// TIA Portal project "PPA-Projekt" (V17)
// Projekt do předmětu PPA

(* hardware
DEVICE "S7-1500/ET200MP station_1"  S7-1500 station
   slot 0: "Rail_0"  Rack  6ES7 590-1***0-0AA0
   slot 1: "PLC_1"  CPU 1516-3 PN/DP  6ES7 516-3AN00-0AB0  V1.8
      slot 3: "CPU display_1"  6ES7591-1BA00-0AA0
      slot 32768: "PROFINET interface_1"  X1
         slot 32769: "Port_1"  X1 P1
         slot 32770: "Port_2"  X1 P2
      slot 33024: "PROFINET interface_2"  X2
         slot 33025: "Port_1"  X2 P1
      slot 33280: "DP interface_1"  X3
DEVICE "HMI_1"  KTP700 Basic PN
   slot 0: "HMI_1"  KTP700 Basic PN  6AV2 123-2GB03-0AX0  17.0.0.0
   slot 1: "HMI_RT_1"  KTP700 Basic PN  6AV2 123-2GB03-0AX0  17.0.0.0
   slot 5: "HMI_1.IE_CP_1"  PROFINET Interface  17.0.0.0
      slot 1: "PROFINET Interface_1"  PROFINET Interface
         slot 1: "Port_1"  Port
*)

// ===== PLC "PLC_1"  CPU 1516-3 PN/DP =====

VAR_GLOBAL   // PLC tag table "Default tag table"
   "SystemInput" AT %MW5 : Int;   // Passed value to PID Setpoints
   "Clock_Byte" AT %MB0 : Byte;
   "Clock_10Hz" AT %M0.0 : Bool;
   "Clock_5Hz" AT %M0.1 : Bool;
   "Clock_2.5Hz" AT %M0.2 : Bool;
   "Clock_2Hz" AT %M0.3 : Bool;
   "Clock_1.25Hz" AT %M0.4 : Bool;
   "Clock_1Hz" AT %M0.5 : Bool;
   "Clock_0.625Hz" AT %M0.6 : Bool;
   "Clock_0.5Hz" AT %M0.7 : Bool;
   "System_Byte" AT %MB1 : Byte;
   "FirstScan" AT %M1.0 : Bool;
   "DiagStatusUpdate" AT %M1.1 : Bool;
   "AlwaysTRUE" AT %M1.2 : Bool;
   "AlwaysFALSE" AT %M1.3 : Bool;
   "SwitchInput" AT %M2.0 : Bool;   // Change SetValue at PID inputs
   "SetValue" AT %MW3 : Int;   // SetValue variable
   "Enable_SystemMatlab" AT %M9.0 : Bool;
   "Enable_SystemTia" AT %M9.1 : Bool;
END_VAR

DATA_BLOCK "LSIM_Matlab"   // DB1
{ S7_Optimized_Access := 'TRUE' }
VERSION : 2.01
// stored: InstanceOfName LSim_PT2aper
"LSim_PT2aper"
BEGIN
END_DATA_BLOCK

DATA_BLOCK "LSIM_TIA"   // DB6
{ S7_Optimized_Access := 'TRUE' }
VERSION : 2.01
// stored: InstanceOfName LSim_PT2aper_1
"LSim_PT2aper_1"
BEGIN
END_DATA_BLOCK

FUNCTION_BLOCK "LSim_PT2aper"   // FB53, SCL
{ S7_Optimized_Access := 'TRUE' }
VERSION : 2.01
   VAR_INPUT
      calcParam : Bool;   // recalculate with new parameters
      input : Real;   // input signal
      tmLag1 : Real := 2.0;   // time constant T1 [sec]
      tmLag2 : Real := 0.2;   // time constant T2 [sec]
      gain : Real := 1.0;   // gain factor
      cycle : Real := 0.1;   // cyclic time [sec]
      maxOut : Real := 100.0;   // max. output limit
      minOut : Real;   // min. output limit
      reset : Bool;   // resets all relevant parameters to ‘0’ including the output
   END_VAR
   VAR_OUTPUT
      error : Bool;   // error (#tmLag1 <= 0 or #tmLag2 <= 0 or #tmLag1 = #tmLag2)
      status : Word;   // status (if #error = TRUE then status = 16#8001)
      maxReached : Bool;   // output has reached max. limit
      minReached : Bool;   // output has reached min. limit
      output : Real;   // output signal (if #error = FALSE)
   END_VAR
   VAR
      statRxn2 : Real;   // delayed input signal (n-2)
      statRxn1 : Real;   // delayed input signal (n-1)
      statRyn2 : Real;   // delayed output signal (n-2)
      statRyn1 : Real;   // delayed output signal (n-1)
      statRf1 : Real;
      statRf2 : Real;
      statRe1 : Real;
      statRe2 : Real;
      statAlpha : Real;
      statBeta : Real;
      statGamma : Real;
      statDelta : Real;
      statOverfirst : Bool;
      statOutput : Real;   // Output signal
   END_VAR
BEGIN
   //=============================================================================
   //SIEMENS AG
   //(c)Copyright 2017 All Rights Reserved
   //-----------------------------------------------------------------------------
   //Library:       Library for Controlled System Simulation
   //Tested with:   S7-1500 FW V2.0 / S7-1200 FW V4.2
   //Engineering:   STEP 7 V14 Upd2 (TIA Portal)
   //Restrictions:  Cyclic interrupt
   //Requirements:  memory card needed for S7-1500
   //Functionality: Simulation of a aperiodic PT2-System
   //  
   //                    gain
   //  F(p) = -----------------------------
   //         (tmLag1*p + 1)*(tmLag2*p + 1)
   //         
   //  Call the simulation in a cyclic interrupt with
   //  cyclic interrupt time at least = tmLag1/10!
   //-----------------------------------------------------------------------------
   //Change log table:
   //Version  Date       Expert in charge                Changes applied
   //02.00.00 03.02.2016 Siemens Industry Online Support Release (STEP 7 V13 SP1)
   //02.00.01 02.03.2017 Siemens Industry Online Support Release (STEP 7 V14)
   //=============================================================================

   // check parameter
   IF #tmLag1 <= 0 OR #tmLag2 <= 0 OR #tmLag1 = #tmLag2 THEN
     #error := TRUE;
     #status := W#16#8001;     // Parameter Error
     #statRxn1 := 0.0;
     #statRyn1 := 0.0;
     #statRxn2 := 0.0;
     #statRyn2 := 0.0;
     #statOutput := 0;
     #output := 0;
     RETURN;
   ELSE
     #error := FALSE;
     #status := W#16#0000;     // no error
   END_IF;

   // calculates the z-parameter for the difference equatation
   IF #calcParam = True OR NOT #statOverfirst THEN
     #statOverfirst := 1;
     // Calculate z-parameters for IT1-System
     #statAlpha := EXP(- #cycle / #tmLag1);
     #statBeta := EXP(- #cycle / #tmLag2);
     #statGamma := #tmLag1 / (#tmLag1 - #tmLag2);
     #statDelta := #tmLag2 / (#tmLag1 - #tmLag2);
     #statRe1 := - #statAlpha - #statBeta;
     #statRe2 := #statAlpha * #statBeta;
     #statRf1 := #gain * (1 - #statGamma * #statAlpha + #statDelta * #statBeta);
     #statRf2 := #gain * (#statAlpha * #statBeta - #statGamma * #statBeta + #statAlpha * #statDelta);
   END_IF;

   // reset Memory
   IF #reset = True THEN
     #statRxn1 := 0.0;
     #statRyn1 := 0.0;
     #statRxn2 := 0.0;
     #statRyn2 := 0.0;
     #statOutput := 0;
   END_IF;
   //save delayed input signals
   #statRxn2 := #statRxn1;
   #statRxn1 := #input;

   //save delayed output signals
   #statRyn2:=#statRyn1;
   #statRyn1:= #statOutput;

   // difference equatation of the PT2-System
   #statOutput := #statRxn1* #statRf1 + #statRxn2*#statRf2 - #statRyn1*#statRe1 - #statRyn2*#statRe2;

   // max limit of acutating variable
   IF #statOutput > #maxOut THEN
     #statOutput := #maxOut;
     #maxReached:= True;
   ELSE
     #maxReached := False;
   END_IF;

   // min limit of acutating variable
   IF #statOutput < #minOut THEN
     #statOutput := #minOut;
     #minReached := True;
   ELSE
     #minReached := False;
   END_IF;

   #output := #statOutput;
END_FUNCTION_BLOCK

FUNCTION_BLOCK "LSim_PT2aper_1"   // FB54, SCL
{ S7_Optimized_Access := 'TRUE' }
VERSION : 2.01
   VAR_INPUT
      calcParam : Bool;   // recalculate with new parameters
      input : Real;   // input signal
      tmLag1 : Real := 2.0;   // time constant T1 [sec]
      tmLag2 : Real := 0.2;   // time constant T2 [sec]
      gain : Real := 1.0;   // gain factor
      cycle : Real := 0.1;   // cyclic time [sec]
      maxOut : Real := 100.0;   // max. output limit
      minOut : Real;   // min. output limit
      reset : Bool;   // resets all relevant parameters to ‘0’ including the output
   END_VAR
   VAR_OUTPUT
      error : Bool;   // error (#tmLag1 <= 0 or #tmLag2 <= 0 or #tmLag1 = #tmLag2)
      status : Word;   // status (if #error = TRUE then status = 16#8001)
      maxReached : Bool;   // output has reached max. limit
      minReached : Bool;   // output has reached min. limit
      output : Real;   // output signal (if #error = FALSE)
   END_VAR
   VAR
      statRxn2 : Real;   // delayed input signal (n-2)
      statRxn1 : Real;   // delayed input signal (n-1)
      statRyn2 : Real;   // delayed output signal (n-2)
      statRyn1 : Real;   // delayed output signal (n-1)
      statRf1 : Real;
      statRf2 : Real;
      statRe1 : Real;
      statRe2 : Real;
      statAlpha : Real;
      statBeta : Real;
      statGamma : Real;
      statDelta : Real;
      statOverfirst : Bool;
      statOutput : Real;   // Output signal
   END_VAR
BEGIN
   //=============================================================================
   //SIEMENS AG
   //(c)Copyright 2017 All Rights Reserved
   //-----------------------------------------------------------------------------
   //Library:       Library for Controlled System Simulation
   //Tested with:   S7-1500 FW V2.0 / S7-1200 FW V4.2
   //Engineering:   STEP 7 V14 Upd2 (TIA Portal)
   //Restrictions:  Cyclic interrupt
   //Requirements:  memory card needed for S7-1500
   //Functionality: Simulation of a aperiodic PT2-System
   //  
   //                    gain
   //  F(p) = -----------------------------
   //         (tmLag1*p + 1)*(tmLag2*p + 1)
   //         
   //  Call the simulation in a cyclic interrupt with
   //  cyclic interrupt time at least = tmLag1/10!
   //-----------------------------------------------------------------------------
   //Change log table:
   //Version  Date       Expert in charge                Changes applied
   //02.00.00 03.02.2016 Siemens Industry Online Support Release (STEP 7 V13 SP1)
   //02.00.01 02.03.2017 Siemens Industry Online Support Release (STEP 7 V14)
   //=============================================================================

   // check parameter
   IF #tmLag1 <= 0 OR #tmLag2 <= 0 OR #tmLag1 = #tmLag2 THEN
     #error := TRUE;
     #status := W#16#8001;     // Parameter Error
     #statRxn1 := 0.0;
     #statRyn1 := 0.0;
     #statRxn2 := 0.0;
     #statRyn2 := 0.0;
     #statOutput := 0;
     #output := 0;
     RETURN;
   ELSE
     #error := FALSE;
     #status := W#16#0000;     // no error
   END_IF;

   // calculates the z-parameter for the difference equatation
   IF #calcParam = True OR NOT #statOverfirst THEN
     #statOverfirst := 1;
     // Calculate z-parameters for IT1-System
     #statAlpha := EXP(- #cycle / #tmLag1);
     #statBeta := EXP(- #cycle / #tmLag2);
     #statGamma := #tmLag1 / (#tmLag1 - #tmLag2);
     #statDelta := #tmLag2 / (#tmLag1 - #tmLag2);
     #statRe1 := - #statAlpha - #statBeta;
     #statRe2 := #statAlpha * #statBeta;
     #statRf1 := #gain * (1 - #statGamma * #statAlpha + #statDelta * #statBeta);
     #statRf2 := #gain * (#statAlpha * #statBeta - #statGamma * #statBeta + #statAlpha * #statDelta);
   END_IF;

   // reset Memory
   IF #reset = True THEN
     #statRxn1 := 0.0;
     #statRyn1 := 0.0;
     #statRxn2 := 0.0;
     #statRyn2 := 0.0;
     #statOutput := 0;
   END_IF;
   //save delayed input signals
   #statRxn2 := #statRxn1;
   #statRxn1 := #input;

   //save delayed output signals
   #statRyn2:=#statRyn1;
   #statRyn1:= #statOutput;

   // difference equatation of the PT2-System
   #statOutput := #statRxn1* #statRf1 + #statRxn2*#statRf2 - #statRyn1*#statRe1 - #statRyn2*#statRe2;

   // max limit of acutating variable
   IF #statOutput > #maxOut THEN
     #statOutput := #maxOut;
     #maxReached:= True;
   ELSE
     #maxReached := False;
   END_IF;

   // min limit of acutating variable
   IF #statOutput < #minOut THEN
     #statOutput := #minOut;
     #minReached := True;
   ELSE
     #minReached := False;
   END_IF;

   #output := #statOutput;
END_FUNCTION_BLOCK

ORGANIZATION_BLOCK "Main"   // OB1, LAD, ProgramCycle
TITLE = "Main Program Sweep (Cycle)"
{ S7_Optimized_Access := 'TRUE' }
VERSION : 0.1
   VAR_INPUT
      Initial_Call : Bool;   // Initial call of this OB
      Remanence : Bool;   // =True, if remanent data are available
   END_VAR
BEGIN
END_ORGANIZATION_BLOCK

ORGANIZATION_BLOCK "Interupt - PID"   // OB30, LAD, CyclicInterrupt
{ S7_Optimized_Access := 'TRUE' }
VERSION : 0.1
   VAR_INPUT
      Initial_Call : Bool;   // Initial call of this OB
      Event_Count : Int;   // Events discarded
   END_VAR
BEGIN

REGION Network 1
   // PID controller - Matlab
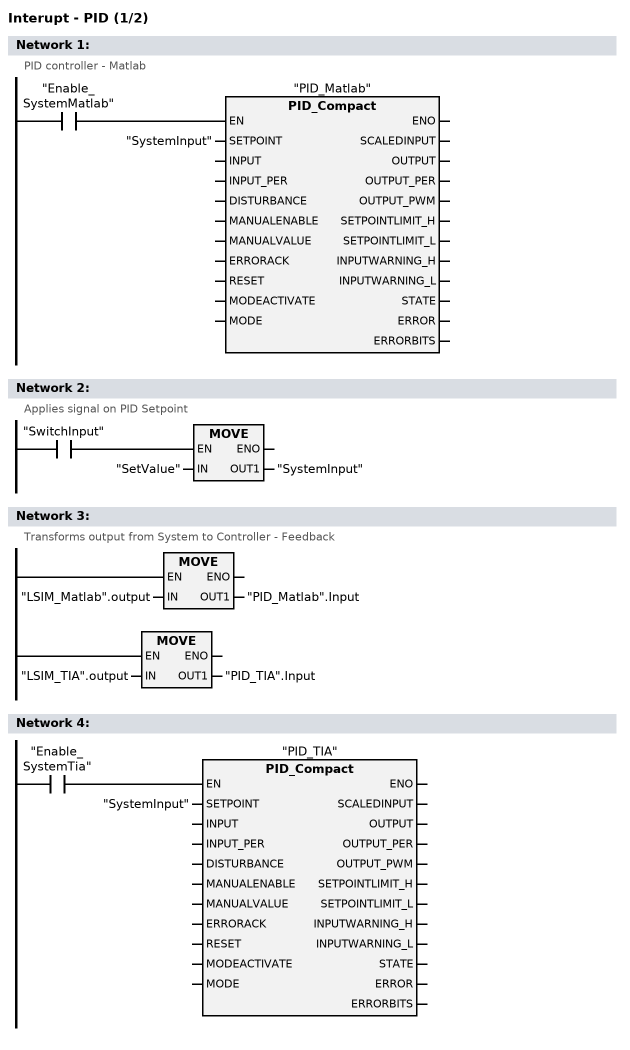
   IF "Enable_SystemMatlab" THEN
       "PID_Matlab"(Setpoint := "SystemInput");   // PID_Compact
   END_IF;
END_REGION

REGION Network 2
   // Applies signal on PID Setpoint
   RUNG wire#powerrail
      Contact( "SwitchInput" )
      Move(in := "SetValue", out1 => "SystemInput")
   END_RUNG
   // the same network as SCL:
   IF "SwitchInput" THEN "SystemInput" := "SetValue"; END_IF;
END_REGION

REGION Network 3
   // Transforms output from System to Controller - Feedback
   RUNG wire#powerrail
      Move(in := "LSIM_Matlab".output, out1 => "PID_Matlab".Input)
   END_RUNG
   RUNG wire#powerrail
      Move(in := "LSIM_TIA".output, out1 => "PID_TIA".Input)
   END_RUNG
   // the same network as SCL:
   "PID_Matlab".Input := "LSIM_Matlab".output;
   "PID_TIA".Input := "LSIM_TIA".output;
END_REGION

REGION Network 4
   IF "Enable_SystemTia" THEN
       "PID_TIA"(Setpoint := "SystemInput");   // PID_Compact
   END_IF;
END_REGION

REGION Network 5
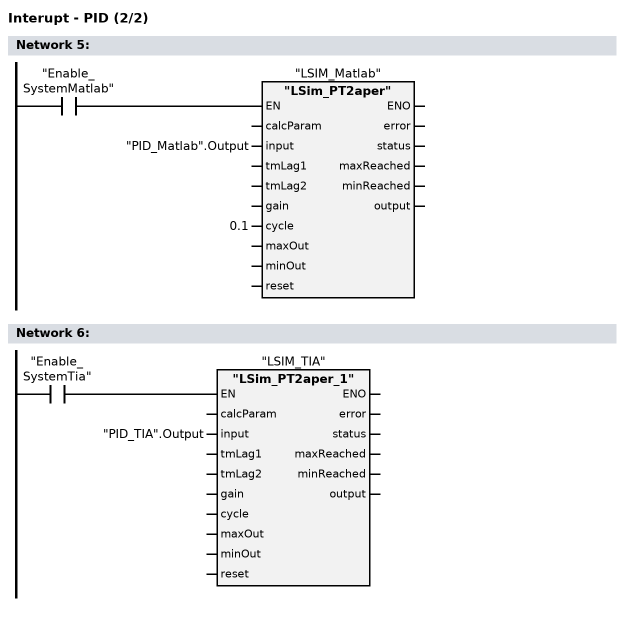
   RUNG wire#powerrail
      Contact( "Enable_SystemMatlab" )
      "LSIM_Matlab"(calcParam :=, input := "PID_Matlab".Output, tmLag1 :=, tmLag2 :=, gain :=, cycle := 0.1, maxOut :=, minOut :=, reset :=, error =>, status =>, maxReached =>, minReached =>, output =>)
   END_RUNG
   // the same network as SCL:
   IF "Enable_SystemMatlab" THEN
       "LSIM_Matlab"(input := "PID_Matlab".Output, cycle := 0.1);   // "LSim_PT2aper"
   END_IF;
END_REGION

REGION Network 6
   RUNG wire#powerrail
      Contact( "Enable_SystemTia" )
      "LSIM_TIA"(calcParam :=, input := "PID_TIA".Output, tmLag1 :=, tmLag2 :=, gain :=, cycle :=, maxOut :=, minOut :=, reset :=, error =>, status =>, maxReached =>, minReached =>, output =>)
   END_RUNG
   // the same network as SCL:
   IF "Enable_SystemTia" THEN
       "LSIM_TIA"(input := "PID_TIA".Output);   // "LSim_PT2aper_1"
   END_IF;
END_REGION
END_ORGANIZATION_BLOCK

ORGANIZATION_BLOCK "Startup"   // OB100, LAD, Startup
TITLE = "Complete Restart"
{ S7_Optimized_Access := 'TRUE' }
VERSION : 0.1
// Intial setup
   VAR_INPUT
      LostRetentive : Bool;   // True if retentive data are lost
      LostRTC : Bool;   // True if date and time are lost
   END_VAR
BEGIN

REGION Network 1
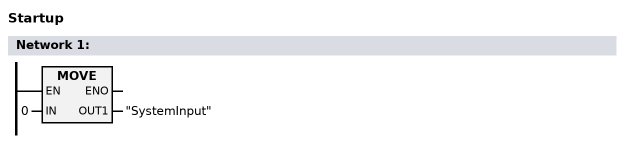
   RUNG wire#powerrail
      Move(in := 0, out1 => "SystemInput")
   END_RUNG
   // the same network as SCL:
   "SystemInput" := 0;
END_REGION
END_ORGANIZATION_BLOCK

(* ===== HMI "HMI_RT_1" =====
system functions are stored by id; their names below are inferred from use
connection "HMI_Connection_1": ETHERNET, SMART_S7_1500_OMS

HMI tags "Default tag table"
   "Tag_ScreenNumber" : UInt, internal
   "LSIM_Matlab_Output" : Real = PLC LSIM_Matlab.output, 100 ms
   "SetValue_Switch" : Bool = PLC SwitchInput AT %M2.0, 100 ms
   "Change_SetValue" : Int = PLC SetValue AT %MW3, 100 ms
   "LSIM_TIA_Output" : Real = PLC LSIM_TIA.output AT %DB1.DBW0, 100 ms
   "System_SetValue" : Int = PLC SystemInput AT %MW5, 100 ms
   "PID_TIA_Output" : Real = PLC PID_TIA.Output, 100 ms
   "PID_Matlab_Output" : Real = PLC PID_Matlab.Output AT %DB1.DBD0, 100 ms
   "Enable_MatlabSystem" : Bool = PLC Enable_SystemMatlab AT %M9.0, 100 ms
   "Enable_TiaSystem" : Bool = PLC Enable_SystemTia AT %M9.1, 100 ms

Template "Template_1" 800x480
   Button "Exit" at 714,429 size 71x50; TextOff 'Exit'; PictureOff "ExitRuntime_KTP700_Basic_PN_TR"; PictureOn "ExitRuntime_KTP700_Basic_PN_TR"
      on Release: StopRuntime(0)
   Button "Template_Button" at 614,429 size 71x50; TextOff 'Text'
   Button "Template_Button_1" at 514,429 size 71x50; TextOff 'Text'
   Button "Template_Button_2" at 414,429 size 71x50; TextOff 'Text'
   Button "Template_Button_3" at 314,429 size 71x50; TextOff 'Text'
   Button "Template_Button_4" at 214,429 size 71x50; TextOff 'Text'
   Button "Alarms" at 114,429 size 71x50; TextOff 'Alarms'; PictureOff "AlarmDisplay_KTP700_Basic_PN_TR"; PictureOn "AlarmDisplay_KTP700_Basic_PN_TR"
      on Release: function_ef3f5d25("Alarm window_Unacknowledged", -1)
   Button "Start screen" at 14,429 size 71x50; TextOff 'Start screen'; PictureOff "NavigateHome_KTP700_Basic_PN_TR"; PictureOn "NavigateHome_KTP700_Basic_PN_TR"
      on Release: ActivateScreen("MainScreen", 0)
   SymbolicIOField "Symbolic_IO_Field_Screen" at 93,9 size 600x33; TextOff '0'; TextOn '1'; TextList "TextList_ScreenNames"
      ProcessValue <- "Tag_ScreenNumber"
      on Change: ActivateScreenByNumber("Tag_ScreenNumber", 0)
   DateTimeField "HmiScreenItemData" at 695,25 size 105x25
   DateTimeField "HmiScreenItemData_1" at 695,0 size 105x25
   GraphicView "Logo" at 0,0 size 91x51; Picture "Logo of HMI_1"

screen "MainScreen" 800x480, template "Template_1"
   on GenerateScreen: SetTag("Tag_ScreenNumber", 1)
   TextField "HmiScreenItemData" at 80,225 size 640x25; Text 'Welcome to HMI_1 (KTP700 Basic+ PN)!'
   TrendView "Trend view_1" at 109,64 size 686x349
   IOField "I/O field_1" at 6,91 size 96x32; FormatPattern s99999
      ProcessValue <- "Change_SetValue"
   TextField "Text field_1" at 8,68 size 97x20; Text 'Set Value (%)'
   Button "Button_1" at 6,133 size 96x94; TextOff 'Set Value'
      on Press: SetTag("SetValue_Switch", 1)
      on Release: SetTag("SetValue_Switch", 0)
   TextField "Text field_2" at 11,129 size 16x23; Text 'Text'
   Switch "Switch_1" at 17,259 size 64x32; CaptionText 'Switch'; TextOff 'OFF'; TextOn 'ON'
      ProcessValue <- "Enable_MatlabSystem"
   TextField "Enable Sys 1" at 5,235 size 100x23; Text 'EN - Matlab'
   Switch "Switch_2" at 17,331 size 64x32; TextOn 'ON'; CaptionText 'Switch'; TextOff 'OFF'
      ProcessValue <- "Enable_TiaSystem"
   TextField "Enable Sys 1_1" at 15,308 size 74x23; Text 'EN - TIA'

screen "PIDOutputs" 800x480, template "Template_1"
   TextField "HmiScreenItemData" at 80,225 size 640x25; Text 'Welcome to HMI_1 (KTP700 Basic+ PN)!'
   TrendView "Trend view_1" at 109,64 size 686x349
   IOField "I/O field_1" at 6,91 size 96x32; FormatPattern s99999
      ProcessValue <- "Change_SetValue"
   TextField "Text field_1" at 8,68 size 97x20; Text 'Set Value (%)'
   Button "Button_1" at 6,133 size 96x94; TextOff 'Set Value'
      on Release: SetTag("SetValue_Switch", 0)
      on Press: SetTag("SetValue_Switch", 1)
   TextField "Text field_2" at 11,129 size 16x23; Text 'Text'
   Switch "Switch_1" at 17,259 size 64x32; TextOn 'ON'; CaptionText 'Switch'; TextOff 'OFF'
      ProcessValue <- "Enable_MatlabSystem"
   Switch "Switch_2" at 17,331 size 64x32; TextOn 'ON'; CaptionText 'Switch'; TextOff 'OFF'
      ProcessValue <- "Enable_TiaSystem"
   TextField "Enable Sys 1_1" at 15,308 size 74x23; Text 'EN - TIA'
   TextField "Enable Sys 1" at 5,235 size 100x23; Text 'EN - Matlab'
*)